FUNCTION_BLOCK Power

VAR_IN_OUT
	state : INT;
END_VAR

VAR
	//Power variable
	Vraw AT %I*	: ARRAY [0 .. Components.system] OF DINT;
	Vsense		: ARRAY [0 .. Components.system] OF REAL;
	Iin			: ARRAY [0 .. Components.system] OF REAL;
	Pin		 	: ARRAY [0 .. Components.system] OF REAL;
	Pin_max		: ARRAY [0 .. Components.system] OF REAL;
	Pin_avg		: ARRAY [0 .. Components.system] OF REAL;
	
	//counter
	i 				: INT;
	powerTotal		: ARRAY [0 .. Components.system] OF REAL;
	powerCounter 	: ARRAY [0 .. Components.system] OF DINT;
	
	//timer
	timer 			: TON;
	timeElapsed		: TIME;
	timer_rtrig		: R_TRIG;
	
	//testvar
	test : INT;
END_VAR

VAR CONSTANT
	Rsense			: REAL := 0.051;
	AdcResolution	: DINT := 8388607; //24bit adc (positive and minus)
	Vin				: ARRAY[0..1] OF REAL := [24.0, 48.0];
	Vref			: REAL := 1.25;
	CountTo			: TIME := T#1000H;
END_VAR

(*This function block is used to monitor shutter system power usage.
The module calculates instantanuous power, average power usage over a motion duration, and max power  *)

//reset power values
IF state=0 THEN
	FOR i := 0 TO Components.system BY 1 DO
		Pin_max[i] := 0;
	END_FOR
END_IF


FOR i:=0 TO (Components.system - 1) BY 1 DO 

//Calculate instantanuous power
	Vsense[i] := (DINT_TO_REAL(Vraw[i])*Vref)/DINT_TO_REAL(AdcResolution);
	Iin[i] := Vsense[i]/Rsense;
	
	IF i=Components.motorXM OR i=Components.motorXP THEN
		Pin[i] := Vin[1]*Iin[i];
	ELSE
		Pin[i] := Vin[0]*Iin[i];
	END_IF

	
//Calculate average power
	IF state <> 100 THEN
		powerTotal[i] := powerTotal[i]+Pin[i];
		powerCounter[i] := powerCounter[i]+1;
		Pin_avg[i] 		:= PowerTotal[i]/DINT_TO_REAL(powerCounter[i]);
	ELSE
			powertotal[i] 	:= 0;
			powerCounter[i]	:= 0;	
	END_IF

	
//Calculate max power
	IF Pin_max[i] < Pin[i] THEN
		Pin_max[i] := Pin[i];
	END_IF
	
END_FOR


//Calculate power of entire shutter
Pin[Components.system] := Pin[Components.motorXP]+Pin[Components.motorXM]+Pin[Components.brakes]
								+ Pin[Components.controller]+Pin[Components.terminals];
Pin_avg[Components.system] := Pin_avg[Components.motorXP]+Pin_avg[Components.motorXM]+Pin_avg[Components.brakes]
								+ Pin_avg[Components.controller]+Pin_avg[Components.terminals];
IF Pin_max[Components.system] < Pin[Components.system] THEN
	Pin_max[Components.system] := Pin[Components.system];
END_IF

END_FUNCTION_BLOCK

(* stored: Version 1.1.0.1, ProductVersion 3.1.4020.12
   POU Power: Id {cd82df6c-11f2-4b61-8c52-0b244f02b6d6}, SpecialFunc None *)
